// TIA Portal V18 export
// export: Created 2026-01-09T11:23:33.1075563Z, ExportSetting WithDefaults, DisplayName Totally Integrated Automation Portal, DisplayVersion V18 Update 5, DisplayName TIA Portal Openness, DisplayVersion V18 Update 5, DisplayName TIA Portal Teamcenter Gateway, DisplayVersion V18, DisplayName TIA Portal Version Control Interface, DisplayVersion V18, DisplayName SINAMICS Startdrive Advanced, DisplayVersion V18 SP2 Update 1, DisplayName SINAMICS Startdrive G110M, G120, G120C, G120D, G120P, G115D, DisplayVersion V18 SP2 Update 1, DisplayName SINAMICS Startdrive G130, G150, S120, S150, SINAMICS MV, S210, G220, S200, DisplayVersion V18 SP2 Update 1, DisplayName STEP 7 Professional, DisplayVersion V18 Update 5, DisplayName STEP 7 Safety, DisplayVersion V18, DisplayName WinCC Professional, DisplayVersion V18 Update 5
Screen "234-Camera_IV3_811A1"  1280x800, Number=234, Template=02ManualUnit1
  ScreenLayer "Layer_0"
    TextField "文本域_25" at 0,83 size 1280x70  Text="工位IV检测 / Manual IV Check / Text"
    FaceplateInstance "HMI_KeyenceCheckerIV3_1" at 0,162 size 1256x532  FaceplateTypeName=03 Function Block@$@Checker@$@ KeyenceCheckerIV3@$@HMI@$@HMI_KeyenceCheckerIV3 V 0.0.8
      KeyenceChecker := DB_KeyenceCheckerIV3_aDev{2}
      ErrorNoList := IV3_ErrorMessages
    Button "btnMenu6" at 640,725 size 128x75  Mode=Text, TextOff="C-IV3相机 811A1 / C-IV3 811A1", TextOn="C-IV3相机 811A1 / C-IV3 811A1"
      on Click: ActivateScreen(Screen name := , Object number := 0)
    Button "btnMenu4" at 384,725 size 128x75  Mode=Text, TextOff="C-三轴伺服 IAI / C-AxisServo IAI", TextOn="C-三轴伺服 IAI / C-AxisServo IAI"
      on Click: ActivateScreen(Screen name := 232_IAIAxis, Object number := 0)
    Button "btnMenu5" at 512,725 size 128x75  Mode=Text, TextOff="C-IV3相机 810A1 / C-IV3 810A1", TextOn="C-IV3相机 810A1 / C-IV3 810A1"
      on Click: ActivateScreen(Screen name := 233-Camera_IV3_810A1, Object number := 0)
    Button "btnMenu7" at 896,725 size 128x75  Mode=Text
    Button "btnMenu7_1" at 1024,725 size 128x75  Mode=Text
    Button "btnMenu6_2" at 768,725 size 128x75  Mode=Text, TextOff="C-涂胶 / C-GlueSys", TextOn="C-涂胶 / C-GlueSys"
      on Click: ActivateScreen(Screen name := 235_Glue, Object number := 0)
    Button "按钮_4" at 128,725 size 128x75  Mode=Text, PictureOff=向右箭头_0, TextOff="C-气缸 / C-Cylinder", TextOn="C-气缸 / C-Cylinder"
      on Click: ActivateScreen(Screen name := 230_Cylinder, Object number := 0)
    Button "btnMenu4_1" at 256,725 size 128x75  Mode=Text, TextOff="C-伺服 382A1 / C-Servo 382A1", TextOn="C-伺服 382A1 / C-Servo 382A1"
      on Click: ActivateScreen(Screen name := 231-Servo_382A1, Object number := 0)
  ScreenLayer "Layer_1"
